// TIA Portal V15.1 export
// export: Created 2024-05-17T05:38:59.5444224Z, ExportSetting WithDefaults, DisplayName Totally Integrated Automation Portal, DisplayVersion V15.1 Update 5, DisplayName TIA Portal Openness, DisplayVersion V15.1 Update 5, DisplayName SINAMICS Startdrive Advanced, DisplayVersion V15.1, DisplayName G130, G150, S120, S150, SINAMICS MV, S210, DisplayVersion V15.1, DisplayName G110M, G120, G120C, G120D, G120P, DisplayVersion V15.1, DisplayName STEP 7 Professional, DisplayVersion V15.1 Update 5, DisplayName STEP 7 Safety, DisplayVersion V15.1, DisplayName WinCC Professional, DisplayVersion V15.1 Update 5, DisplayName SIMATIC Visualization Architect, DisplayVersion V15.1
FUNCTION "209000NCP01Passiv" : Void   // FC252, FBD
TITLE = 209000NCP01Passiv
{ S7_Optimized_Access := 'FALSE' }
AUTHOR : VCC
NAME : LocFunc
VERSION : 0.1
// stored: AutoNumber false, IsIECCheckEnabled false, SetENOAutomatically False, UDAEnableTagReadback false
   VAR_OUTPUT
      O_AlarmA : Bool;   // Alarm A
      O_AlarmB : Bool;   // Alarm B
      O_AlarmC : Bool;   // Alarm C
      O_AlarmD : Bool;   // Alarm D
      O_AlarmABCondition : Bool;   // Alarms resetable
      H_IAnim : Word;   // Icon Animation
   END_VAR
   VAR_TEMP
      TEMP0 : Bool;
   END_VAR
BEGIN

REGION Network 1: **** 1 - Inputs **** HMI Reset Passivation
   // HMI Reset Passivation
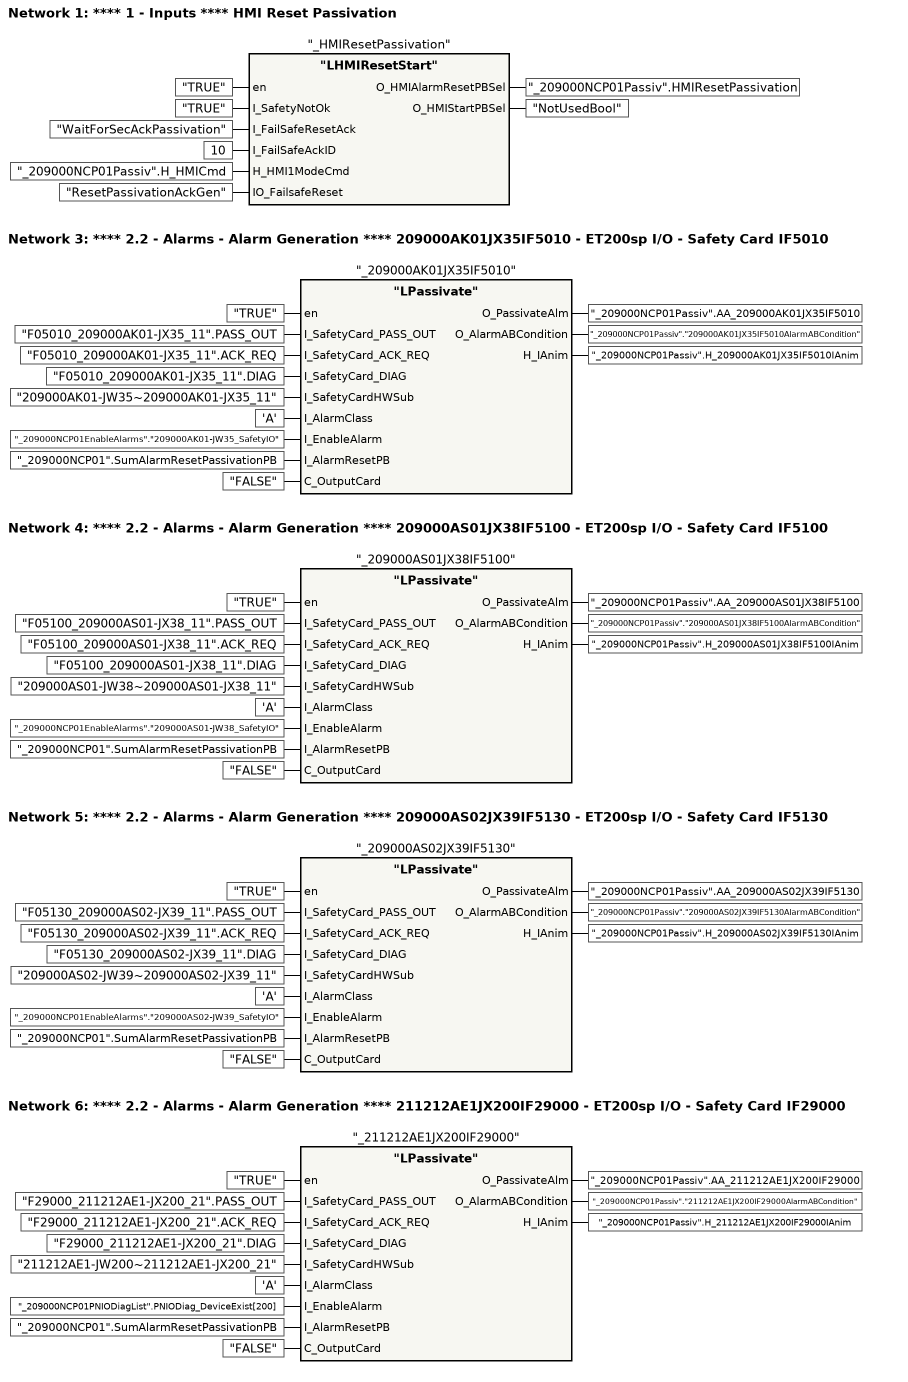
   IF "TRUE" THEN
       "_HMIResetPassivation"(I_SafetyNotOk := "TRUE",   // "LHMIResetStart"
                              I_FailSafeResetAck := "WaitForSecAckPassivation",
                              I_FailSafeAckID := 10,
                              H_HMI1ModeCmd := "_209000NCP01Passiv".H_HMICmd,
                              IO_FailsafeReset := "ResetPassivationAckGen",
                              O_HMIAlarmResetPBSel => "_209000NCP01Passiv".HMIResetPassivation,
                              O_HMIStartPBSel => "NotUsedBool");
   END_IF;
END_REGION

REGION Network 2: **** --------------------- ET200sp I/O --------------------- ****
END_REGION

REGION Network 3: **** 2.2 - Alarms - Alarm Generation **** 209000AK01JX35IF5010 - ET200sp I/O - Safety Card IF5010
   // Passivation alarm - ET200sp I/O - Safety Card IF5010
   IF "TRUE" THEN
       "_209000AK01JX35IF5010"(I_SafetyCard_PASS_OUT := "F05010_209000AK01-JX35_11".PASS_OUT,   // "LPassivate"
                               I_SafetyCard_ACK_REQ := "F05010_209000AK01-JX35_11".ACK_REQ,
                               I_SafetyCard_DIAG := "F05010_209000AK01-JX35_11".DIAG,
                               I_SafetyCardHWSub := "209000AK01-JW35~209000AK01-JX35_11",
                               I_AlarmClass := 'A',
                               I_EnableAlarm := "_209000NCP01EnableAlarms"."209000AK01-JW35_SafetyIO",
                               I_AlarmResetPB := "_209000NCP01".SumAlarmResetPassivationPB,
                               C_OutputCard := "FALSE",
                               O_PassivateAlm => "_209000NCP01Passiv".AA_209000AK01JX35IF5010,
                               O_AlarmABCondition => "_209000NCP01Passiv"."209000AK01JX35IF5010AlarmABCondition",
                               H_IAnim => "_209000NCP01Passiv".H_209000AK01JX35IF5010IAnim);
   END_IF;
END_REGION

REGION Network 4: **** 2.2 - Alarms - Alarm Generation **** 209000AS01JX38IF5100 - ET200sp I/O - Safety Card IF5100
   // Passivation alarm - ET200sp I/O - Safety Card IF5100
   IF "TRUE" THEN
       "_209000AS01JX38IF5100"(I_SafetyCard_PASS_OUT := "F05100_209000AS01-JX38_11".PASS_OUT,   // "LPassivate"
                               I_SafetyCard_ACK_REQ := "F05100_209000AS01-JX38_11".ACK_REQ,
                               I_SafetyCard_DIAG := "F05100_209000AS01-JX38_11".DIAG,
                               I_SafetyCardHWSub := "209000AS01-JW38~209000AS01-JX38_11",
                               I_AlarmClass := 'A',
                               I_EnableAlarm := "_209000NCP01EnableAlarms"."209000AS01-JW38_SafetyIO",
                               I_AlarmResetPB := "_209000NCP01".SumAlarmResetPassivationPB,
                               C_OutputCard := "FALSE",
                               O_PassivateAlm => "_209000NCP01Passiv".AA_209000AS01JX38IF5100,
                               O_AlarmABCondition => "_209000NCP01Passiv"."209000AS01JX38IF5100AlarmABCondition",
                               H_IAnim => "_209000NCP01Passiv".H_209000AS01JX38IF5100IAnim);
   END_IF;
END_REGION

REGION Network 5: **** 2.2 - Alarms - Alarm Generation **** 209000AS02JX39IF5130 - ET200sp I/O - Safety Card IF5130
   // Passivation alarm - ET200sp I/O - Safety Card IF5130
   IF "TRUE" THEN
       "_209000AS02JX39IF5130"(I_SafetyCard_PASS_OUT := "F05130_209000AS02-JX39_11".PASS_OUT,   // "LPassivate"
                               I_SafetyCard_ACK_REQ := "F05130_209000AS02-JX39_11".ACK_REQ,
                               I_SafetyCard_DIAG := "F05130_209000AS02-JX39_11".DIAG,
                               I_SafetyCardHWSub := "209000AS02-JW39~209000AS02-JX39_11",
                               I_AlarmClass := 'A',
                               I_EnableAlarm := "_209000NCP01EnableAlarms"."209000AS02-JW39_SafetyIO",
                               I_AlarmResetPB := "_209000NCP01".SumAlarmResetPassivationPB,
                               C_OutputCard := "FALSE",
                               O_PassivateAlm => "_209000NCP01Passiv".AA_209000AS02JX39IF5130,
                               O_AlarmABCondition => "_209000NCP01Passiv"."209000AS02JX39IF5130AlarmABCondition",
                               H_IAnim => "_209000NCP01Passiv".H_209000AS02JX39IF5130IAnim);
   END_IF;
END_REGION

REGION Network 6: **** 2.2 - Alarms - Alarm Generation **** 211212AE1JX200IF29000 - ET200sp I/O - Safety Card IF29000
   // Passivation alarm - ET200sp I/O - Safety Card IF29000
   IF "TRUE" THEN
       "_211212AE1JX200IF29000"(I_SafetyCard_PASS_OUT := "F29000_211212AE1-JX200_21".PASS_OUT,   // "LPassivate"
                               I_SafetyCard_ACK_REQ := "F29000_211212AE1-JX200_21".ACK_REQ,
                               I_SafetyCard_DIAG := "F29000_211212AE1-JX200_21".DIAG,
                               I_SafetyCardHWSub := "211212AE1-JW200~211212AE1-JX200_21",
                               I_AlarmClass := 'A',
                               I_EnableAlarm := "_209000NCP01PNIODiagList".PNIODiag_DeviceExist[200],
                               I_AlarmResetPB := "_209000NCP01".SumAlarmResetPassivationPB,
                               C_OutputCard := "FALSE",
                               O_PassivateAlm => "_209000NCP01Passiv".AA_211212AE1JX200IF29000,
                               O_AlarmABCondition => "_209000NCP01Passiv"."211212AE1JX200IF29000AlarmABCondition",
                               H_IAnim => "_209000NCP01Passiv".H_211212AE1JX200IF29000IAnim);
   END_IF;
END_REGION

REGION Network 7: **** 2.2 - Alarms - Alarm Generation **** 211212AE1JX200IF29006 - ET200sp I/O - Safety Card IF29006
   // Passivation alarm - ET200sp I/O - Safety Card IF29006
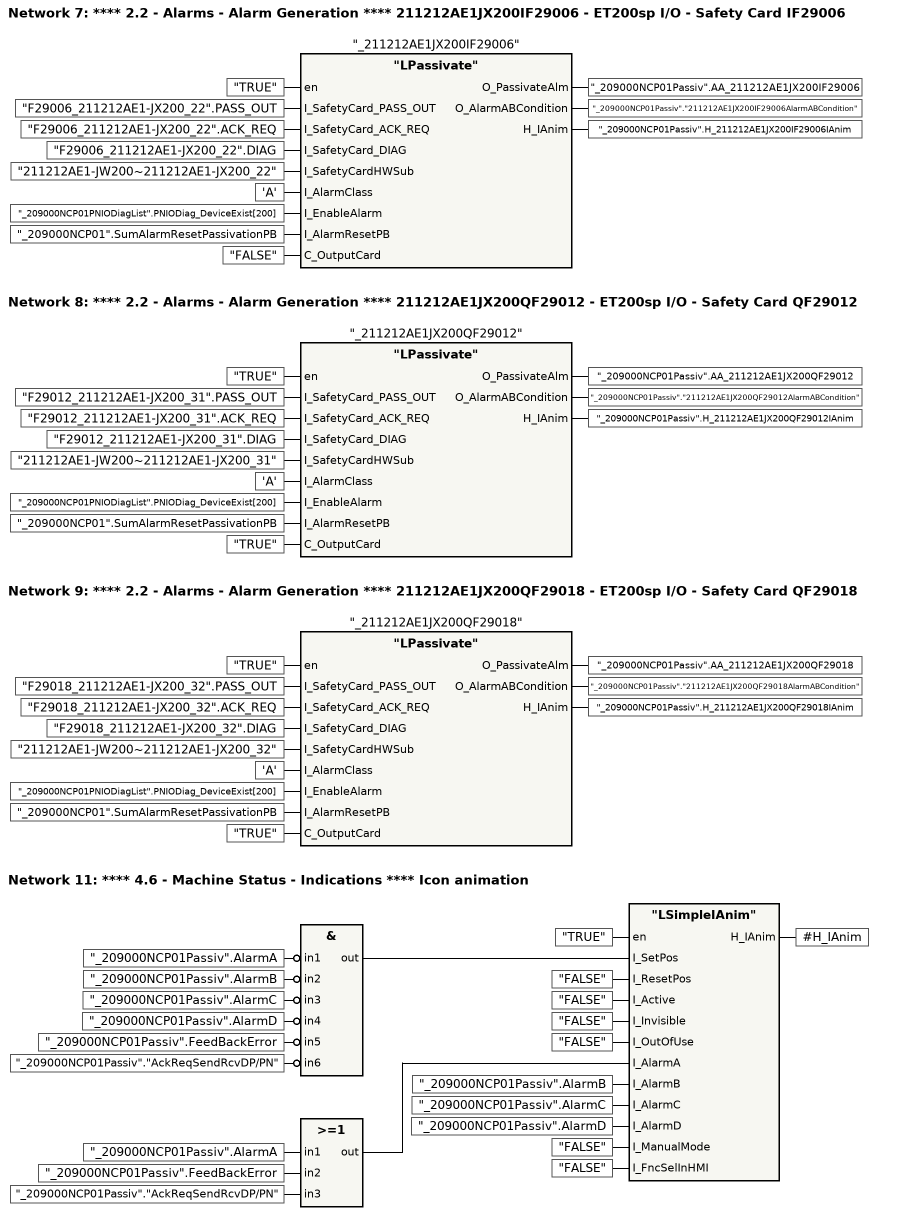
   IF "TRUE" THEN
       "_211212AE1JX200IF29006"(I_SafetyCard_PASS_OUT := "F29006_211212AE1-JX200_22".PASS_OUT,   // "LPassivate"
                               I_SafetyCard_ACK_REQ := "F29006_211212AE1-JX200_22".ACK_REQ,
                               I_SafetyCard_DIAG := "F29006_211212AE1-JX200_22".DIAG,
                               I_SafetyCardHWSub := "211212AE1-JW200~211212AE1-JX200_22",
                               I_AlarmClass := 'A',
                               I_EnableAlarm := "_209000NCP01PNIODiagList".PNIODiag_DeviceExist[200],
                               I_AlarmResetPB := "_209000NCP01".SumAlarmResetPassivationPB,
                               C_OutputCard := "FALSE",
                               O_PassivateAlm => "_209000NCP01Passiv".AA_211212AE1JX200IF29006,
                               O_AlarmABCondition => "_209000NCP01Passiv"."211212AE1JX200IF29006AlarmABCondition",
                               H_IAnim => "_209000NCP01Passiv".H_211212AE1JX200IF29006IAnim);
   END_IF;
END_REGION

REGION Network 8: **** 2.2 - Alarms - Alarm Generation **** 211212AE1JX200QF29012 - ET200sp I/O - Safety Card QF29012
   // Passivation alarm - ET200sp I/O - Safety Card QF29012
   IF "TRUE" THEN
       "_211212AE1JX200QF29012"(I_SafetyCard_PASS_OUT := "F29012_211212AE1-JX200_31".PASS_OUT,   // "LPassivate"
                               I_SafetyCard_ACK_REQ := "F29012_211212AE1-JX200_31".ACK_REQ,
                               I_SafetyCard_DIAG := "F29012_211212AE1-JX200_31".DIAG,
                               I_SafetyCardHWSub := "211212AE1-JW200~211212AE1-JX200_31",
                               I_AlarmClass := 'A',
                               I_EnableAlarm := "_209000NCP01PNIODiagList".PNIODiag_DeviceExist[200],
                               I_AlarmResetPB := "_209000NCP01".SumAlarmResetPassivationPB,
                               C_OutputCard := "TRUE",
                               O_PassivateAlm => "_209000NCP01Passiv".AA_211212AE1JX200QF29012,
                               O_AlarmABCondition => "_209000NCP01Passiv"."211212AE1JX200QF29012AlarmABCondition",
                               H_IAnim => "_209000NCP01Passiv".H_211212AE1JX200QF29012IAnim);
   END_IF;
END_REGION

REGION Network 9: **** 2.2 - Alarms - Alarm Generation **** 211212AE1JX200QF29018 - ET200sp I/O - Safety Card QF29018
   // Passivation alarm - ET200sp I/O - Safety Card QF29018
   IF "TRUE" THEN
       "_211212AE1JX200QF29018"(I_SafetyCard_PASS_OUT := "F29018_211212AE1-JX200_32".PASS_OUT,   // "LPassivate"
                               I_SafetyCard_ACK_REQ := "F29018_211212AE1-JX200_32".ACK_REQ,
                               I_SafetyCard_DIAG := "F29018_211212AE1-JX200_32".DIAG,
                               I_SafetyCardHWSub := "211212AE1-JW200~211212AE1-JX200_32",
                               I_AlarmClass := 'A',
                               I_EnableAlarm := "_209000NCP01PNIODiagList".PNIODiag_DeviceExist[200],
                               I_AlarmResetPB := "_209000NCP01".SumAlarmResetPassivationPB,
                               C_OutputCard := "TRUE",
                               O_PassivateAlm => "_209000NCP01Passiv".AA_211212AE1JX200QF29018,
                               O_AlarmABCondition => "_209000NCP01Passiv"."211212AE1JX200QF29018AlarmABCondition",
                               H_IAnim => "_209000NCP01Passiv".H_211212AE1JX200QF29018IAnim);
   END_IF;
END_REGION

REGION Network 10: **** -------------------------------------------------- ****
END_REGION

REGION Network 11: **** 4.6 - Machine Status - Indications **** Icon animation
   // Icon animation
   IF "TRUE" THEN
       "LSimpleIAnim"(I_SetPos := NOT "_209000NCP01Passiv".AlarmA AND NOT "_209000NCP01Passiv".AlarmB AND NOT "_209000NCP01Passiv".AlarmC AND NOT "_209000NCP01Passiv".AlarmD AND NOT "_209000NCP01Passiv".FeedBackError AND NOT "_209000NCP01Passiv"."AckReqSendRcvDP/PN",
                      I_ResetPos := "FALSE",
                      I_Active := "FALSE",
                      I_Invisible := "FALSE",
                      I_OutOfUse := "FALSE",
                      I_AlarmA := "_209000NCP01Passiv".AlarmA OR "_209000NCP01Passiv".FeedBackError OR "_209000NCP01Passiv"."AckReqSendRcvDP/PN",
                      I_AlarmB := "_209000NCP01Passiv".AlarmB,
                      I_AlarmC := "_209000NCP01Passiv".AlarmC,
                      I_AlarmD := "_209000NCP01Passiv".AlarmD,
                      I_ManualMode := "FALSE",
                      I_FncSelInHMI := "FALSE",
                      H_IAnim => #H_IAnim);
   END_IF;
END_REGION

REGION Network 12: **** 4.6 - Machine status - Indications **** Animation
   // Animation
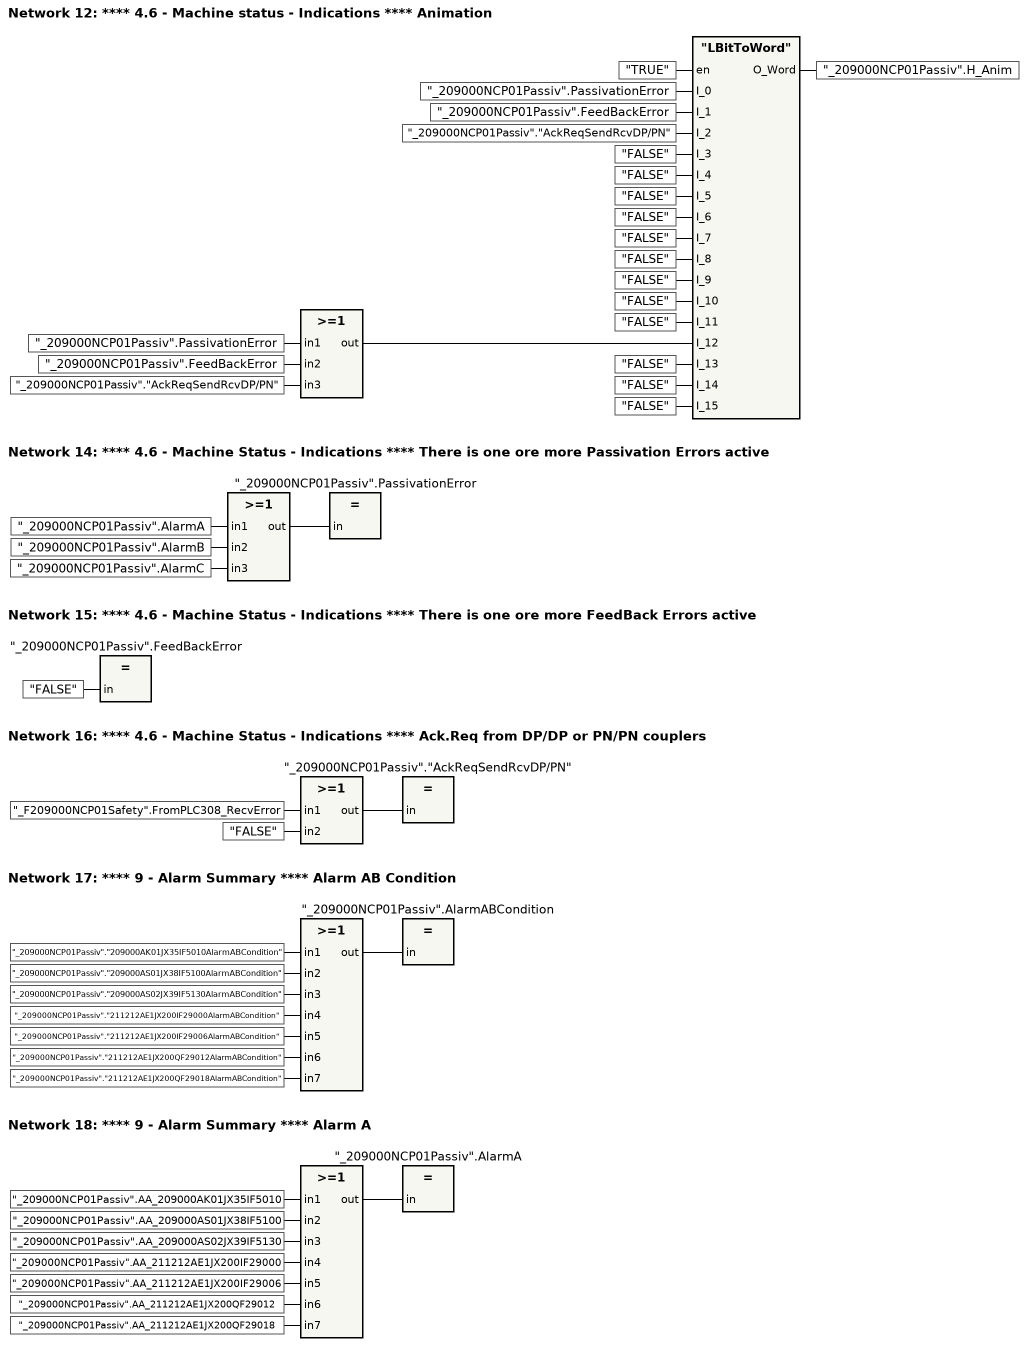
   IF "TRUE" THEN
       "LBitToWord"(I_0 := "_209000NCP01Passiv".PassivationError,
                    I_1 := "_209000NCP01Passiv".FeedBackError,
                    I_2 := "_209000NCP01Passiv"."AckReqSendRcvDP/PN",
                    I_3 := "FALSE",
                    I_4 := "FALSE",
                    I_5 := "FALSE",
                    I_6 := "FALSE",
                    I_7 := "FALSE",
                    I_8 := "FALSE",
                    I_9 := "FALSE",
                    I_10 := "FALSE",
                    I_11 := "FALSE",
                    I_12 := "_209000NCP01Passiv".PassivationError OR "_209000NCP01Passiv".FeedBackError OR "_209000NCP01Passiv"."AckReqSendRcvDP/PN",
                    I_13 := "FALSE",
                    I_14 := "FALSE",
                    I_15 := "FALSE",
                    O_Word => "_209000NCP01Passiv".H_Anim);
   END_IF;
END_REGION

NETWORK
TITLE = **** 4.6 - Machine Status - Indications **** Animation DB number
// DB number
      OPN   "_209000NCP01Passiv";
      L     DBNO;
      T     "_209000NCP01Passiv".H_DBnr;

REGION Network 14: **** 4.6 - Machine Status - Indications **** There is one ore more Passivation Errors active
   // There is one ore more Passivation Errors active
   "_209000NCP01Passiv".PassivationError := "_209000NCP01Passiv".AlarmA OR "_209000NCP01Passiv".AlarmB OR "_209000NCP01Passiv".AlarmC;
END_REGION

REGION Network 15: **** 4.6 - Machine Status - Indications **** There is one ore more FeedBack Errors active
   // There is one ore more FeedBack Errors active
   "_209000NCP01Passiv".FeedBackError := "FALSE";
END_REGION

REGION Network 16: **** 4.6 - Machine Status - Indications **** Ack.Req from DP/DP or PN/PN couplers
   // Ack.Req from DP/DP or PN/PN couplers
   "_209000NCP01Passiv"."AckReqSendRcvDP/PN" := "_F209000NCP01Safety".FromPLC308_RecvError OR "FALSE";
END_REGION

REGION Network 17: **** 9 - Alarm Summary **** Alarm AB Condition
   // Alarm AB condition for the general Profinet
   "_209000NCP01Passiv".AlarmABCondition := "_209000NCP01Passiv"."209000AK01JX35IF5010AlarmABCondition" OR "_209000NCP01Passiv"."209000AS01JX38IF5100AlarmABCondition" OR "_209000NCP01Passiv"."209000AS02JX39IF5130AlarmABCondition" OR "_209000NCP01Passiv"."211212AE1JX200IF29000AlarmABCondition" OR "_209000NCP01Passiv"."211212AE1JX200IF29006AlarmABCondition" OR "_209000NCP01Passiv"."211212AE1JX200QF29012AlarmABCondition" OR "_209000NCP01Passiv"."211212AE1JX200QF29018AlarmABCondition";
END_REGION

REGION Network 18: **** 9 - Alarm Summary **** Alarm A
   // Summary of alarms A
   "_209000NCP01Passiv".AlarmA := "_209000NCP01Passiv".AA_209000AK01JX35IF5010 OR "_209000NCP01Passiv".AA_209000AS01JX38IF5100 OR "_209000NCP01Passiv".AA_209000AS02JX39IF5130 OR "_209000NCP01Passiv".AA_211212AE1JX200IF29000 OR "_209000NCP01Passiv".AA_211212AE1JX200IF29006 OR "_209000NCP01Passiv".AA_211212AE1JX200QF29012 OR "_209000NCP01Passiv".AA_211212AE1JX200QF29018;
END_REGION

REGION Network 19: **** 9 - Alarm Summary **** Alarm B
   // Summary of alarms B
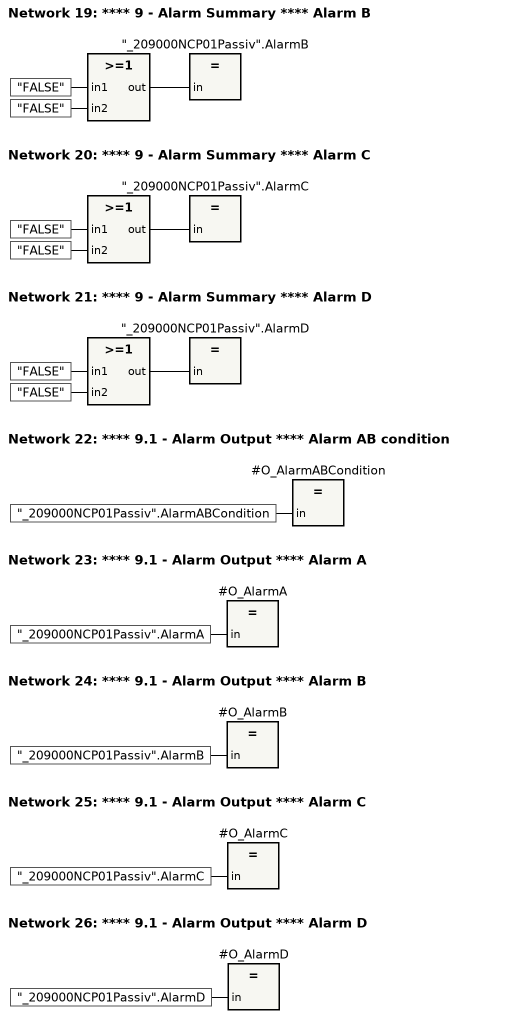
   "_209000NCP01Passiv".AlarmB := "FALSE" OR "FALSE";
END_REGION

REGION Network 20: **** 9 - Alarm Summary **** Alarm C
   // Summary of alarms C
   "_209000NCP01Passiv".AlarmC := "FALSE" OR "FALSE";
END_REGION

REGION Network 21: **** 9 - Alarm Summary **** Alarm D
   // Summary of alarms D
   "_209000NCP01Passiv".AlarmD := "FALSE" OR "FALSE";
END_REGION

REGION Network 22: **** 9.1 - Alarm Output **** Alarm AB condition
   // Alarm AB condition
   #O_AlarmABCondition := "_209000NCP01Passiv".AlarmABCondition;
END_REGION

REGION Network 23: **** 9.1 - Alarm Output **** Alarm A
   // Output Alarm A
   #O_AlarmA := "_209000NCP01Passiv".AlarmA;
END_REGION

REGION Network 24: **** 9.1 - Alarm Output **** Alarm B
   // Output Alarm B
   #O_AlarmB := "_209000NCP01Passiv".AlarmB;
END_REGION

REGION Network 25: **** 9.1 - Alarm Output **** Alarm C
   // Output Alarm C
   #O_AlarmC := "_209000NCP01Passiv".AlarmC;
END_REGION

REGION Network 26: **** 9.1 - Alarm Output **** Alarm D
   // Output Alarm D
   #O_AlarmD := "_209000NCP01Passiv".AlarmD;
END_REGION

REGION Network 27: **** 9.2 - Alarm DWord**** Alarm To DWord
   // Alarm Word
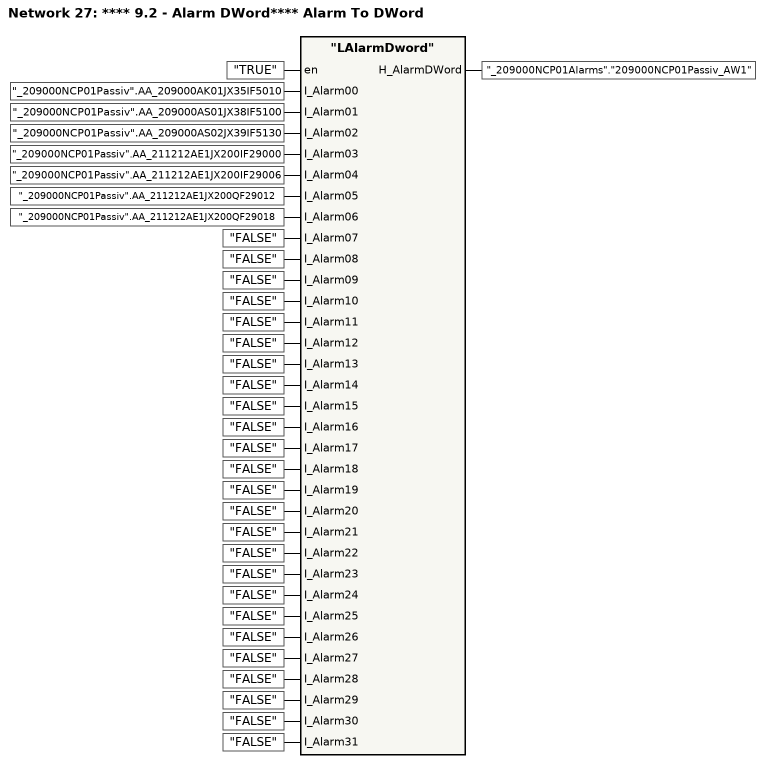
   IF "TRUE" THEN
       "LAlarmDword"(I_Alarm00 := "_209000NCP01Passiv".AA_209000AK01JX35IF5010,
                     I_Alarm01 := "_209000NCP01Passiv".AA_209000AS01JX38IF5100,
                     I_Alarm02 := "_209000NCP01Passiv".AA_209000AS02JX39IF5130,
                     I_Alarm03 := "_209000NCP01Passiv".AA_211212AE1JX200IF29000,
                     I_Alarm04 := "_209000NCP01Passiv".AA_211212AE1JX200IF29006,
                     I_Alarm05 := "_209000NCP01Passiv".AA_211212AE1JX200QF29012,
                     I_Alarm06 := "_209000NCP01Passiv".AA_211212AE1JX200QF29018,
                     I_Alarm07 := "FALSE",
                     I_Alarm08 := "FALSE",
                     I_Alarm09 := "FALSE",
                     I_Alarm10 := "FALSE",
                     I_Alarm11 := "FALSE",
                     I_Alarm12 := "FALSE",
                     I_Alarm13 := "FALSE",
                     I_Alarm14 := "FALSE",
                     I_Alarm15 := "FALSE",
                     I_Alarm16 := "FALSE",
                     I_Alarm17 := "FALSE",
                     I_Alarm18 := "FALSE",
                     I_Alarm19 := "FALSE",
                     I_Alarm20 := "FALSE",
                     I_Alarm21 := "FALSE",
                     I_Alarm22 := "FALSE",
                     I_Alarm23 := "FALSE",
                     I_Alarm24 := "FALSE",
                     I_Alarm25 := "FALSE",
                     I_Alarm26 := "FALSE",
                     I_Alarm27 := "FALSE",
                     I_Alarm28 := "FALSE",
                     I_Alarm29 := "FALSE",
                     I_Alarm30 := "FALSE",
                     I_Alarm31 := "FALSE",
                     H_AlarmDWord => "_209000NCP01Alarms"."209000NCP01Passiv_AW1");
   END_IF;
END_REGION
END_FUNCTION
